# B&R Automation Studio project ACPtrak_Widget
Automation Studio 4.7.4.67 SP; technology packages: mappControl 5.11.0, mappMotion 5.11.2, mappView 5.11.2

## Configuration Simulation

CPU PC_any, AutomationRuntime A4.73, Build 4.1.2, Safety 0.0, Vc V4.62.0

### Task classes (Cpu.sw)
```
Cyclic#1 (cycle 400 us, tolerance 0 us):
  Main <- Main.prg
  WidgetData <- WidgetData.prg
Cyclic#2 (cycle 2000 us, tolerance 0 us):
  Vis <- Vis.prg
DataObjects: McAcpSys
Binaries: McAcpSim, FWRules, udbdef, McAcpDrv, arsvcreg, TCData, McProfGen, mvLoader, Config_1, Config_2, Config_4, ashwd, ashwac, asfw, iomap, sysconf, Config_3, Role, User, arconfig, Config_5, Config_6, Config_7, Config_8
Libraries: McBase, McAxis, McAcpTrak, McPureVAx, MpAxis, MpBase, TrakKit, standard, AsBrStr, McAcpAx, AsMath, FileIO, runtime, MTBasics, brsystem, MTTypes, sys_lib, powerlnk, astime, asieccon, arssl, asepl
```

### Hardware
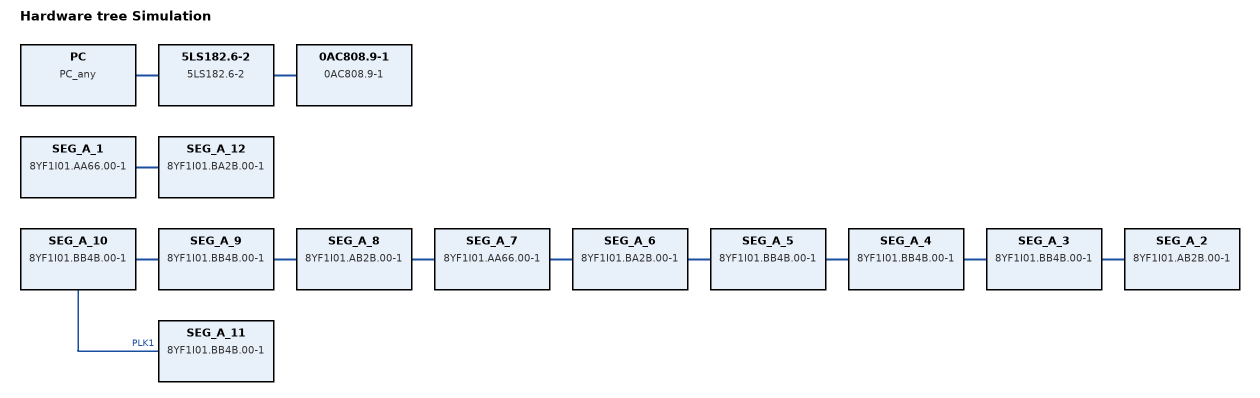
```
0AC808.9-1 : 0AC808.9-1 v1.0.0.0  [ETH1 -> 5LS182.6-2.IF1 [Cable Type=PowerlinkCable, Length=10, Version=1.0.0.2]; ETH2 -> SEG_A_1.PLK3 [Cable Type=PowerlinkCable, Length=10, Version=1.0.0.2]]
5LS182.6-2 : 5LS182.6-2 v1.4.0.0  [SL -> PC.SL2]
PC : PC_any v1.1.0.0 (OrderNumber=PC)
  ConfigurationID = StarwheelSim_Simulation
  VolatileGlobalPvSize = 132000
  SystemTick = 400
  Cyclic1Duration = 400
  Cyclic1Tolerance = 0
  Cyclic2Duration = 2000
  Cyclic2Tolerance = 0
  FileDevice1
  FileDeviceName1 = SvgData
  FileDevicePath1 = ../../../../Logical/Visuals
  FileDevice2
  FileDeviceName2 = User
  FileDevicePath2 = C:\ACPtrak\TeslaStarwheel\TrakPower
  ActivateOpcUa = 1
  OpcUaInformationModels_PV_Version = 1
SEG_A_1 : 8YF1I01.AA66.00-1 v0.0.0.3  [PLK1 -> SEG_A_2.PLK2 [Cable Type=PowerlinkCable, Length=10, Version=1.0.0.2]; PLK2 -> SEG_A_12.PLK1 [Cable Type=PowerlinkCable, Length=10, Version=1.0.0.2]; PLK3 -> 0AC808.9-1.ETH2 [Cable Type=PowerlinkCable, Length=10, Version=1.0.0.2]]
  DriveConfiguration:
    McTypeID = LLMConfig
  DriveConfiguration/Segment:
    Shape = STRAIGHT660
    SegmentReference = SEG_A_1
    StopReaction = UseAssemblySetting
    SpeedFilter = UseAssemblySetting
SEG_A_10 : 8YF1I01.BB4B.00-1 v0.0.0.3  [PLK1 -> SEG_A_11.PLK2 [Cable Type=PowerlinkCable, Length=10, Version=1.0.0.2]; PLK2 -> SEG_A_9.PLK1 [Cable Type=PowerlinkCable, Length=10, Version=1.0.0.2]]
  DriveConfiguration/Segment:
    SegmentReference = ::SEG_A_10
SEG_A_11 : 8YF1I01.BB4B.00-1 v0.0.0.3  [PLK2 -> SEG_A_10.PLK1 [Cable Type=PowerlinkCable, Length=10, Version=1.0.0.2]]
  DriveConfiguration/Segment:
    SegmentReference = ::SEG_A_11
SEG_A_12 : 8YF1I01.BA2B.00-1 v0.0.0.3  [PLK1 -> SEG_A_1.PLK2 [Cable Type=PowerlinkCable, Length=10, Version=1.0.0.2]]
  DriveConfiguration/Segment:
    SegmentReference = ::SEG_A_12
SEG_A_2 : 8YF1I01.AB2B.00-1 v0.0.0.3  [PLK1 -> SEG_A_3.PLK2 [Cable Type=PowerlinkCable, Length=10, Version=1.0.0.2]; PLK2 -> SEG_A_1.PLK1 [Cable Type=PowerlinkCable, Length=10, Version=1.0.0.2]]
  DriveConfiguration/Segment:
    SegmentReference = ::SEG_A_2
SEG_A_3 : 8YF1I01.BB4B.00-1 v0.0.0.3  [PLK1 -> SEG_A_4.PLK2 [Cable Type=PowerlinkCable, Length=10, Version=1.0.0.2]; PLK2 -> SEG_A_2.PLK1 [Cable Type=PowerlinkCable, Length=10, Version=1.0.0.2]]
  DriveConfiguration/Segment:
    SegmentReference = ::SEG_A_3
SEG_A_4 : 8YF1I01.BB4B.00-1 v0.0.0.3  [PLK1 -> SEG_A_5.PLK2 [Cable Type=PowerlinkCable, Length=10, Version=1.0.0.2]; PLK2 -> SEG_A_3.PLK1 [Cable Type=PowerlinkCable, Length=10, Version=1.0.0.2]]
  DriveConfiguration/Segment:
    SegmentReference = ::SEG_A_4
SEG_A_5 : 8YF1I01.BB4B.00-1 v0.0.0.3  [PLK1 -> SEG_A_6.PLK2 [Cable Type=PowerlinkCable, Length=10, Version=1.0.0.2]; PLK2 -> SEG_A_4.PLK1 [Cable Type=PowerlinkCable, Length=10, Version=1.0.0.2]]
  DriveConfiguration/Segment:
    SegmentReference = ::SEG_A_5
SEG_A_6 : 8YF1I01.BA2B.00-1 v0.0.0.3  [PLK1 -> SEG_A_7.PLK2 [Cable Type=PowerlinkCable, Length=10, Version=1.0.0.2]; PLK2 -> SEG_A_5.PLK1 [Cable Type=PowerlinkCable, Length=10, Version=1.0.0.2]]
  DriveConfiguration/Segment:
    SegmentReference = ::SEG_A_6
SEG_A_7 : 8YF1I01.AA66.00-1 v0.0.0.3  [PLK1 -> SEG_A_8.PLK2 [Cable Type=PowerlinkCable, Length=10, Version=1.0.0.2]; PLK2 -> SEG_A_6.PLK1 [Cable Type=PowerlinkCable, Length=10, Version=1.0.0.2]]
  DriveConfiguration/Segment:
    SegmentReference = ::SEG_A_7
SEG_A_8 : 8YF1I01.AB2B.00-1 v0.0.0.3  [PLK1 -> SEG_A_9.PLK2 [Cable Type=PowerlinkCable, Length=10, Version=1.0.0.2]; PLK2 -> SEG_A_7.PLK1 [Cable Type=PowerlinkCable, Length=10, Version=1.0.0.2]]
  DriveConfiguration/Segment:
    SegmentReference = ::SEG_A_8
SEG_A_9 : 8YF1I01.BB4B.00-1 v0.0.0.3  [PLK1 -> SEG_A_10.PLK2 [Cable Type=PowerlinkCable, Length=10, Version=1.0.0.2]; PLK2 -> SEG_A_8.PLK1 [Cable Type=PowerlinkCable, Length=10, Version=1.0.0.2]]
  DriveConfiguration/Segment:
    SegmentReference = ::SEG_A_9
```

### Config_1.assembly - PC/mappMotion/Config_1.assembly
```
Element gAssembly_1 (Type=assembly)
  Tracks:
    TrackSeparation = 0.030
    Track[1]:
      Segments:
        SegmentRef[1] = ::SEG_A_1
        SegmentRef[2] = ::SEG_A_2
        SegmentRef[3] = ::SEG_A_3
        SegmentRef[4] = ::SEG_A_4
        SegmentRef[5] = ::SEG_A_5
        SegmentRef[6] = ::SEG_A_6
        SegmentRef[7] = ::SEG_A_7
        SegmentRef[8] = ::SEG_A_8
        SegmentRef[9] = ::SEG_A_9
        SegmentRef[10] = ::SEG_A_10
        SegmentRef[11] = ::SEG_A_11
        SegmentRef[12] = ::SEG_A_12
      Position = Absolute
        SegmentCountDirection = RightToLeft
        Translation:
          X = 0.0
          Y = 0.0
          Z = 0.0
        Orientation:
          Angle1 = 0.0
          Angle2 = 0.0
          Angle3 = 180
  CommonSegmentSettings:
    SegmentSimulationOnPLC = Off
    StopReaction = InductionHalt
    SpeedFilter = NotUsed
    ControllerParameters:
      DefaultParameter:
        Controller:
          Position:
            ProportionalGain = 0.0
          Speed:
            ProportionalGain = 0.0
            IntegrationTime = 0.0
          FeedForward:
            TotalMass = 0.0
            ForcePositive = 0.0
            ForceNegative = 0.0
            SpeedForceFactor = 0.0
            ForceLoad = 0.0
        MovementErrorLimits:
          PositionError = 0.0
          VelocityError = 0.0
      AdditionalParameterSets = NotUsed
  Shuttles:
    MaxShuttleCount = 50
    ShuttleStereotypes:
      ShuttleStRef[1] = ShuttleStereotype_1
    MagnetPlateConfigurations:
      ShuttleType[1] = 8F1SA.102.xxxxxx-x
    CollisionAvoidance:
      Strategy = Constant
      MaximumModelDimensions:
        Length:
          ExtentToFront = 0.025
          ExtentToBack = 0.025
        Width:
          Width = 0.030
  Visualization:
    MonitoringPv = ::gShuttleMon
    ProcessingTaskClass = 2
```

### Config_2.shuttlestereotype - PC/mappMotion/Config_2.shuttlestereotype
```
Element ShuttleStereotype_1 (Type=shuttlestereotype)
  MeasurementUnit = 5067858
  MeasurementResolution = 0.00001
  MovementLimits = Internal
    VelocityIsReadOnly = 0
    Velocity:
      Velocity = 4.0
    AccelerationIsReadOnly = 0
    Acceleration:
      Acceleration = 50
    DecelerationIsReadOnly = 0
    Deceleration:
      Deceleration = 50
  JerkFilter = Used
    JerkTime = 0.02
  UserData:
    Size = 8
```

### Config_3.sector - PC/mappMotion/Config_3.sector
```
Element Sector_Spawn (Type=sector)
  Type = Composed
    StartSegment:
      SegmentRef = ::SEG_A_7
      Position = 0.33
      PositionRelativeTo = FromEnd
    EndSegment:
      SegmentRef = ::SEG_A_7
Element Sector_Infeed (Type=sector)
  Type = Composed
    StartSegment:
      SegmentRef = ::SEG_A_2
    IntermediateSegments:
      SegmentRef[1] = ::SEG_A_1
      SegmentRef[2] = ::SEG_A_12
      SegmentRef[3] = ::SEG_A_11
      SegmentRef[4] = ::SEG_A_10
      SegmentRef[5] = ::SEG_A_9
    EndSegment:
      SegmentRef = ::SEG_A_8
```

### Config_4.processpointlist - PC/mappMotion/Config_4.processpointlist
```
Element List_PP_Spawn (Type=processpointlist)
  ProcessPoint[0]:
    Name = PP_Spawn_In
    SectorRef = Sector_Spawn
    TriggerEventBufferSize = 10
    BarrierFunctionality = On
  ProcessPoint[1]:
    Name = PP_Spawn_Out
    SectorRef = Sector_Spawn
    PositionRelativeTo = FromEnd
    TriggerEventBufferSize = 10
    BarrierFunctionality = Off
Element List_PP_Outfeed (Type=processpointlist)
  ProcessPoint[0]:
    Name = PP_Outfeed_Sync
    SectorRef = Sector_Outfeed
    Position = 0.165
    TriggerEventBufferSize = 10
    BarrierFunctionality = Off
  ProcessPoint[1]:
    Name = PP_Outfeed_Release
    SectorRef = Sector_Outfeed
    Position = 0.57
    PositionRelativeTo = FromEnd
    TriggerEventBufferSize = 10
    BarrierFunctionality = Off
Element List_PP_Infeed (Type=processpointlist)
  ProcessPoint[0]:
    Name = PP_Infeed_Sync
    SectorRef = Sector_Infeed
    Position = 0.45
    TriggerEventBufferSize = 10
    BarrierFunctionality = On
  ProcessPoint[1]:
    Name = PP_Infeed_Release
    SectorRef = Sector_Infeed
    Position = 0.465
    PositionRelativeTo = FromEnd
    TriggerEventBufferSize = 10
    BarrierFunctionality = Off
```

### Config_5.axis - PC/mappMotion/InfeedAxis/Config_5.axis
```
Element gAxis_1 (Type=axis)
  BaseTypeIsReadOnly = 0
  BaseType = RotaryPeriodic
    MeasurementUnitIsReadOnly = 0
    MeasurementUnit = 17476
    MeasurementResolutionIsReadOnly = 0
    MeasurementResolution = 0.001
    CountDirectionIsReadOnly = 0
    CountDirection = Standard
    PeriodSettings:
      Period = 360.0
  MovementLimitsIsReadOnly = 0
  MovementLimits = Internal
    Position:
      LowerLimitMin = -1.79769313486231E308
      UpperLimitMax = 1.79769313486231E308
      LowerLimit = -1000.0
      UpperLimit = 1000.0
    VelocityIsReadOnly = 0
    Velocity:
      VelocityMax = 3.4E38
      Velocity = 720.0
    AccelerationIsReadOnly = 0
    Acceleration:
      AccelerationMax = 3.4E38
      Acceleration = 720.0
    DecelerationIsReadOnly = 0
    Deceleration:
      DecelerationMax = 3.4E38
      Deceleration = 720.0
  Alarms = None
```

### Config_6.purevaxcfg - PC/mappMotion/InfeedAxis/Config_6.purevaxcfg
```
Element PureVAxCfg_1 (Type=purevaxcfg)
  TypeID = PureVAxConfig
  PureVAxis:
    AxisReference = gAxis_1
```

## Logical view

Binary libraries used (declarations not repeated): operator, runtime, astime, AsIecCon, standard, AsBrStr, AsMath, FileIO, brsystem, MTTypes 1.03.4, sys_lib, McBase 5.11.2, McPureVAx 5.11.2, McAcpAx 5.11.2, McAcpTrak 5.11.2, McAxis 5.11.2, MpAxis 5.11.2, MpBase 5.11.0, MTBasics 5.11.0

### Global.typ - Global data types
```iecst
TYPE
	SyncObj_typ : 	STRUCT
		MoveCyclic : MC_BR_ElasticMoveCycPos_AcpTrak;
		InSync : BOOL;
		PocketSelect : USINT;
		ThisShuttle : McAxisType;
		PeriodSelect : USINT;
		LastCycleSetpoint : LREAL;
	END_STRUCT;
	UserData_typ : 	STRUCT
		SyncObjectID : UINT;
		Color : enumUserColor;
	END_STRUCT;
	TrakCmd_typ : 	STRUCT
		PowerOn : BOOL;
	END_STRUCT;
	TrakPar_typ : 	STRUCT
		Acceleration : REAL;
		Velocity : REAL;
		PPM : REAL;
	END_STRUCT;
	TrakStatus_typ : 	STRUCT
		State : USINT;
	END_STRUCT;
	Trak_typ : 	STRUCT
		Cmd : TrakCmd_typ;
		Par : TrakPar_typ;
		Status : TrakStatus_typ;
	END_STRUCT;
	Reference_typ : 	STRUCT
		PosRad : REAL;
		PosDeg : REAL;
	END_STRUCT;
	Period_typ : 	STRUCT
		Pocket : ARRAY[0..MAX_NUM_POCKETS]OF Pockets_typ;
		PocketLastCycle : ARRAY[0..MAX_NUM_POCKETS]OF Pockets_typ;
		TrakMax : REAL;
		TrakMin : REAL;
	END_STRUCT;
	Starwheel_typ : 	STRUCT
		Axis : MpAxisBasic;
		Period : ARRAY[0..MAX_NUM_PERIODS]OF Period_typ;
	END_STRUCT;
	Pockets_typ : 	STRUCT
		Offset : REAL;
		PosDeg : REAL;
		PosRad : REAL;
		TrakPos : LREAL;
	END_STRUCT;
	ProcessPoint_typ : 	STRUCT
		RoutedMoveVel : MC_BR_RoutedMoveVel_AcpTrak;
		TrgEnable : MC_BR_TrgPointEnable_AcpTrak;
		TrgInfo : MC_BR_TrgPointGetInfo_AcpTrak;
		ShUserData : MC_BR_ShCopyUserData_AcpTrak;
		UserDataBuffer : UserData_typ;
		Counter : UDINT;
		State : USINT;
		BarrierCmd : MC_BR_BarrierCommand_AcpTrak;
		BarrierReadInfo : MC_BR_BarrierReadInfo_AcpTrak;
		BarrierState : USINT;
		periodSelect : USINT;
		pocketSelect : USINT;
	END_STRUCT;
	StarSectorPar_typ : 	STRUCT
		R1 : REAL;
		R2 : REAL;
		deltaT : TIME;
		SectorTangentPos : REAL;
		PocketCount : USINT;
		Wm : REAL;
		ReleaseVelocity : REAL;
		PositionSyncPP : REAL;
		Rp : REAL;
		PeriodCount : USINT;
		PositionRelPP : REAL;
	END_STRUCT;
	StarwheelSectorLogic_typ : 	STRUCT
		Starwheel : Starwheel_typ;
		SyncPP : ProcessPoint_typ;
		ReleasePP : ProcessPoint_typ;
		SyncObj : ARRAY[0..NUM_SYNC_OBJS]OF SyncObj_typ;
		indexOpenSyncObj : USINT;
		Par : StarSectorPar_typ;
	END_STRUCT;
END_TYPE
```

### Segments.var - Global variables
```iecst
VAR
	SEG_A_1 : McSegmentType;
	SEG_A_2 : McSegmentType;
	SEG_A_3 : McSegmentType;
	SEG_A_4 : McSegmentType;
	SEG_A_5 : McSegmentType;
	SEG_A_6 : McSegmentType;
	SEG_A_7 : McSegmentType;
	SEG_A_8 : McSegmentType;
	SEG_A_9 : McSegmentType;
	SEG_A_10 : McSegmentType;
	SEG_A_11 : McSegmentType;
	SEG_A_12 : McSegmentType;
END_VAR
```

### Global.var - Global variables
```iecst
VAR
	gShuttleMon : McAcpTrakAssemblyMonData;
	gTrak : Trak_typ;
END_VAR
VAR CONSTANT
	NUM_SYNC_OBJS : USINT := 20;
	MAX_NUM_POCKETS : USINT := 16;
END_VAR
VAR
	Infeed : StarwheelSectorLogic_typ;
END_VAR
VAR CONSTANT
	MAX_NUM_PERIODS : USINT := 5;
END_VAR
```

### Package Logical/Libraries - Global libraries

### Library Logical/Libraries/TrakKit (IEC)

#### Types.typ - Exported data types
```iecst
TYPE
	enumUserColor :
		(
		GRAY,
		BLUE,
		RED,
		GREEN,
		YELLOW,
		ORANGE,
		WHITE,
		BLACK,
		PINK,
		PURPLE
		);
	typShuttleUserData : 	STRUCT
		Color : enumUserColor;
		SyncObjectID : UINT;
		InSync : BOOL;
	END_STRUCT;
	ClearBlockState :
		(
		CLEAR_BLOCK_STATE_IDLE,
		CLEAR_BLOCK_STATE_INIT,
		CLEAR_BLOCK_STATE_WAIT,
		CLEAR_BLOCK_STATE_RESET,
		CLEAR_BLOCK_STATE_OFF
		);
	ClearPPState :
		(
		CLEAR_PP_STATE_IDLE,
		CLEAR_PP_STATE_ENABLE,
		CLEAR_PP_STATE_WAIT,
		CLEAR_PP_STATE_GET_INFO,
		CLEAR_PP_STATE_OFF
		);
	SpawnState :
		(
		SPAWN_STATE_IDLE,
		SPAWN_STATE_BLOCK,
		SPAWN_STATE_CREATE,
		SPAWN_STATE_REPORT,
		SPAWN_STATE_CREATE_NEXT,
		SPAWN_STATE_GET,
		SPAWN_STATE_SET_USER_DATA,
		SPAWN_STATE_SEND,
		SPAWN_STATE_WAIT,
		SPAWN_STATE_TRIG,
		SPAWN_STATE_UNBLOCK,
		SPAWN_STATE_DONE
		);
	FeedState :
		(
		FEED_STATE_IDLE,
		FEED_STATE_ENABLE,
		FEED_STATE_WAIT,
		FEED_STATE_TRIG,
		FEED_STATE_CHECK_SHUTTLE,
		FEED_STATE_GET_SHUTTLE_DATA,
		FEED_STATE_MOVE_ABS,
		FEED_STATE_TIME,
		FEED_STATE_GET,
		FEED_STATE_COLOR,
		FEED_STATE_SEND,
		FEED_STATE_DISABLE
		);
	TwoUpState1 :
		(
		TWOUP_STATE1_IDLE,
		TWOUP_STATE1_ENABLE,
		TWOUP_STATE1_WAIT,
		TWOUP_STATE1_TRIG,
		TWOUP_STATE1_CHECK_SHUTTLE,
		TWOUP_STATE1_MOVE_ABS,
		TWOUP_STATE1_TIME,
		TWOUP_STATE1_DISABLE
		);
	TwoUpState2 :
		(
		TWOUP_STATE2_IDLE,
		TWOUP_STATE2_WAIT,
		TWOUP_STATE2_GET1,
		TWOUP_STATE2_MOVE_ABS,
		TWOUP_STATE2_TIME,
		TWOUP_STATE2_GET2,
		TWOUP_STATE2_COLOR,
		TWOUP_STATE2_SEND
		);
END_TYPE
```

#### TrakKit.fun - Exported functions and function blocks
```iecst
FUNCTION_BLOCK ShuttleSpawn
	VAR_INPUT
		Enable : BOOL;
		StartPP : UDINT; (*Process point at start to block any incoming shuttle*)
		EndPP : UDINT; (*Process point at end to check shuttles have left*)
		Sector : UDINT; (*Sector to create shuttles on*)
		SectorPositionStart : LREAL; (*Position to start creating shuttles*)
		SectorPositionIncrement : LREAL; (*Increment to create shuttles*)
		DstSector : DINT; (*Destination Sector*)
		DstSectorPosition : LREAL; (*Destination sector position*)
		Velocity : REAL; (*Velocity of move*)
		RouteVelocity : REAL;
		Acceleration : {REDUND_UNREPLICABLE} REAL; (*Acceleration of move*)
		NumShuttleBatch : USINT; (*Number of shuttles in a batch*)
		NumShuttleTotal : USINT; (*Total shuttles to spawn*)
		SetShuttleData : MC_BR_ShCopyUserData_AcpTrak;
		AcknSpawn : BOOL;
	END_VAR
	VAR_OUTPUT
		SpawnValid : BOOL;
		SpawnedAxis : McAxisType;
		Done : BOOL;
	END_VAR
	VAR
		InternalSectorPositionStart : LREAL;
		InternalSectorPositionIncrement : LREAL;
		InternalNumShuttleBatch : USINT;
		InternalNumShuttleTotal : USINT;
		ExitShuttleNum : USINT; (*Number of shuttles that have left*)
		BatchCreated : USINT; (*Number of shuttles created in the batch*)
		TotalCreated : USINT; (*Number of shuttles created total*)
		State : SpawnState;
		TrigEnable : MC_BR_TrgPointEnable_AcpTrak;
		TrigInfo : MC_BR_TrgPointGetInfo_AcpTrak;
		Barrier : MC_BR_BarrierCommand_AcpTrak;
		AddShuttle : MC_BR_SecAddShuttle_AcpTrak;
		GetShuttle : MC_BR_SecGetShuttle_AcpTrak;
		MoveVel : MC_BR_RoutedMoveVel_AcpTrak;
		InternalUserData : typShuttleUserData;
	END_VAR
END_FUNCTION_BLOCK

FUNCTION_BLOCK ShuttleDelete
END_FUNCTION_BLOCK

FUNCTION_BLOCK Redirect
END_FUNCTION_BLOCK

FUNCTION_BLOCK Feed
	VAR_INPUT
		Enable : BOOL;
		PP : UDINT;
		NumShuttles : USINT;
		Sector : UDINT;
		UseAbsMove : BOOL;
		UseVelMoveTrigger : BOOL;
		VelMovTrigger : BOOL;
		SectorPositionStart : LREAL;
		TrigDirection : McAcpTrakTrgPointEventEnum;
		MoveAbsVelocity : REAL;
		SectorPositionIncrement : LREAL;
		DstSector : UDINT;
		DstSectorPosition : LREAL;
		DstStartDirection : McDirectionEnum;
		Color : enumUserColor;
		Velocity : REAL;
		RouteVelocity : REAL;
		Acceleration : REAL;
		FeedTime : TIME;
	END_VAR
	VAR_OUTPUT
		Done : BOOL;
		ReadyForProduct : BOOL;
	END_VAR
	VAR
		InternalNumShuttles : USINT;
		InternalSectorPositionStart : LREAL;
		InternalSectorPositionIncrement : LREAL;
		InternalUserData : typShuttleUserData;
		LastSeqNumber : UDINT;
		LastShuttleNumber : USINT;
		ShuttleCount : USINT;
		State : FeedState;
		TrigEnable : MC_BR_TrgPointEnable_AcpTrak;
		TrigInfo : MC_BR_TrgPointGetInfo_AcpTrak;
		CheckShuttle : MC_BR_ShReadInfo_AcpTrak;
		MoveAbs : MC_BR_RoutedMoveAbs_AcpTrak;
		GetShuttle : MC_BR_SecGetShuttle_AcpTrak;
		ColorShuttle : MC_BR_ShCopyUserData_AcpTrak;
		MoveVel : MC_BR_RoutedMoveVel_AcpTrak;
		FeedTON : TON;
		ReadShuttleData : MC_BR_ShCopyUserData_AcpTrak;
	END_VAR
END_FUNCTION_BLOCK

FUNCTION_BLOCK ClearArea
	VAR_INPUT
		Enable : BOOL;
		StartPP : UDINT;
		EndPP : UDINT;
		NumShuttles : USINT; (*Number of shuttles to allow*)
		newParam : BOOL;
	END_VAR
	VAR
		ExitShuttleNum : USINT; (*Number of shuttles that have left*)
		BlockState : ClearBlockState;
		PPState : ClearPPState;
		TrigEnable : MC_BR_TrgPointEnable_AcpTrak;
		TrigInfo : MC_BR_TrgPointGetInfo_AcpTrak;
		Barrier : MC_BR_BarrierCommand_AcpTrak;
	END_VAR
END_FUNCTION_BLOCK

FUNCTION_BLOCK CalculatePPM
	VAR_INPUT
		Enable : BOOL;
		PP : UDINT;
		NumberOfShuttlesToAvg : LREAL; (*Max 10000*)
		TrigDirection : McAcpTrakTrgPointEventEnum;
	END_VAR
	VAR_OUTPUT
		PPM : LREAL;
	END_VAR
	VAR
		FinishedLoadout : BOOL;
		LastSeqNumber : UDINT;
		ShuttlesPassed : INT;
		TotalShuttlesPassed : UDINT;
		TimeTotal : UDINT;
		TimeStart : ARRAY[0..10000] OF DATE_AND_TIME;
		TimeDelta : UDINT;
		State : UINT;
		TrigEnable : MC_BR_TrgPointEnable_AcpTrak;
		TrigInfo : MC_BR_TrgPointGetInfo_AcpTrak;
		CheckShuttle : MC_BR_ShReadInfo_AcpTrak;
		DTGetTime_0 : DTGetTime;
		LastTimeDeltaIndex : UINT;
	END_VAR
END_FUNCTION_BLOCK

FUNCTION_BLOCK TwoUp
	VAR_INPUT
		Enable : BOOL;
		PP : UDINT;
		NumShuttles : USINT;
		Sector : ARRAY[0..1] OF UDINT;
		SectorPositionStart : ARRAY[0..1] OF LREAL;
		SectorPositionIncrement : ARRAY[0..1] OF LREAL;
		DstSector : UDINT;
		DstSectorPosition : LREAL;
		Color : enumUserColor;
		Velocity : REAL;
		Acceleration : REAL;
		FeedTime : ARRAY[0..1] OF TIME;
	END_VAR
	VAR
		InternalNumShuttles : USINT;
		InternalPosArray : ARRAY[0..8] OF LREAL;
		InternalSectorPositionStart : ARRAY[0..1] OF LREAL;
		InternalSectorPositionIncrement : ARRAY[0..1] OF LREAL;
		InternalUserData : typShuttleUserData;
		ShuttleCount : USINT;
		State1 : TwoUpState1;
		State2 : TwoUpState2;
		TrigEnable : MC_BR_TrgPointEnable_AcpTrak;
		TrigInfo : MC_BR_TrgPointGetInfo_AcpTrak;
		CheckShuttle : MC_BR_ShReadInfo_AcpTrak;
		MoveAbs : ARRAY[0..1] OF MC_BR_RoutedMoveAbs_AcpTrak;
		GetShuttle : ARRAY[0..1] OF MC_BR_SecGetShuttle_AcpTrak;
		MoveVel : MC_BR_RoutedMoveVel_AcpTrak;
		ColorShuttle : MC_BR_ShCopyUserData_AcpTrak;
		FeedTON : ARRAY[0..1] OF TON;
		Increment : BOOL; (*Increment from first to second segment*)
	END_VAR
END_FUNCTION_BLOCK
```

#### ShuttleSpawn.st
```iecst
FUNCTION_BLOCK ShuttleSpawn

	CASE State OF

		SPAWN_STATE_IDLE:

			IF Enable THEN
				InternalSectorPositionStart := SectorPositionStart;
				InternalSectorPositionIncrement := SectorPositionIncrement;
				InternalNumShuttleTotal := NumShuttleTotal;
				InternalNumShuttleBatch := NumShuttleBatch;
				//				InternalUserData.ShuttleNumber := 0;
				//				InternalUserData.Color := BLUE;
			//	InternalUserData.FirstShuttle := 1;
				TrigEnable.ProcessPoint := EndPP;
				TrigEnable.Enable := 1;
				TrigInfo.ProcessPoint := EndPP;
				Barrier.ProcessPoint := StartPP;
				Barrier.Command := mcACPTRAK_BARRIER_CLOSE;
				Barrier.Execute := 1;
				AddShuttle.Sector := Sector;
				AddShuttle.AdvancedParameters.Velocity := Velocity;
				AddShuttle.Position := InternalSectorPositionStart;
				GetShuttle.Sector := Sector;
				GetShuttle.Mode := mcACPTRAK_SEARCH_FORWARD;
//  added F.Forthuber
				SpawnValid := FALSE;
//  end
				SetShuttleData.Axis  := ADR(GetShuttle.Axis);
				SetShuttleData.DataAddress := ADR(InternalUserData);
				SetShuttleData.DataSize := SIZEOF(InternalUserData);
				SetShuttleData.Mode := mcACPTRAK_USERDATA_SET;
				MoveVel.Axis := ADR(GetShuttle.Axis);
				MoveVel.Sector := DstSector;
				MoveVel.Position := DstSectorPosition;
				MoveVel.Velocity := Velocity;
				MoveVel.RouteVelocity := RouteVelocity;
				MoveVel.Acceleration := Acceleration;
				MoveVel.Deceleration := Acceleration;
				MoveVel.AdvancedParameters.StartDirection := mcDIR_POSITIVE;
				MoveVel.AdvancedParameters.EndDirection := mcDIR_POSITIVE;
				MoveVel.AdvancedParameters.ShuttleOrientation := mcDIR_UNDEFINED;
				State := SPAWN_STATE_BLOCK;
			END_IF

		SPAWN_STATE_BLOCK:

			IF TrigEnable.Valid AND Barrier.Done THEN
				Barrier.Execute := 0;
				AddShuttle.Execute := 1;
				Done:=FALSE;
				State := SPAWN_STATE_CREATE;
			END_IF

		SPAWN_STATE_CREATE:

			IF AddShuttle.Done THEN
//  added F.Forthuber
				SpawnedAxis := AddShuttle.Axis;
				SpawnValid:=TRUE;
				State := SPAWN_STATE_REPORT;
			END_IF

		SPAWN_STATE_REPORT:

			IF AcknSpawn THEN
				SpawnValid:=FALSE;
//  end
				BatchCreated := BatchCreated + 1;
				TotalCreated := TotalCreated + 1;
				AddShuttle.Execute := 0;
				IF (BatchCreated >= InternalNumShuttleBatch) OR (TotalCreated >= InternalNumShuttleTotal) THEN
					BatchCreated := 0;
					GetShuttle.Enable := 1;
					State := SPAWN_STATE_GET;
				ELSE
					State := SPAWN_STATE_CREATE_NEXT;
				END_IF
			END_IF

		SPAWN_STATE_CREATE_NEXT:

			AddShuttle.Position := AddShuttle.Position + InternalSectorPositionIncrement;
			AddShuttle.Execute := 1;
			State := SPAWN_STATE_CREATE;

		SPAWN_STATE_GET:

			IF GetShuttle.Valid THEN
				GetShuttle.Next := 0;
				//InternalUserData.ShuttleNumber := InternalUserData.ShuttleNumber + 1;
				SetShuttleData.Execute := 1;
				State := SPAWN_STATE_SET_USER_DATA;
			END_IF

		SPAWN_STATE_SET_USER_DATA:
			IF SetShuttleData.Done THEN
				SetShuttleData.Execute := 0;
				MoveVel.Execute := 1;
				State := SPAWN_STATE_SEND;
			END_IF;

		SPAWN_STATE_SEND:

			IF MoveVel.Active THEN
	//			InternalUserData.FirstShuttle := 0;
				MoveVel.Execute := 0;
				IF GetShuttle.RemainingCount = 0 THEN
					GetShuttle.Enable := 0;
					State := SPAWN_STATE_WAIT;
				ELSE
					GetShuttle.Next := 1;
					State := SPAWN_STATE_GET;
				END_IF
			END_IF

		SPAWN_STATE_WAIT:

			IF NOT Enable  THEN
				TotalCreated := 0;
				ExitShuttleNum := 0;
				TrigEnable.Enable := 0;
				Barrier.Command := mcACPTRAK_BARRIER_OPEN;
				Barrier.Execute := 1;
				State := SPAWN_STATE_UNBLOCK;
			ELSIF TotalCreated >= InternalNumShuttleTotal THEN
				TotalCreated := 0;
				TrigEnable.Enable := 0;
				Barrier.Command := mcACPTRAK_BARRIER_OPEN;
				Barrier.Execute := 1;
				State := SPAWN_STATE_UNBLOCK;
			ELSIF ExitShuttleNum >= InternalNumShuttleBatch THEN
				ExitShuttleNum := 0;
				AddShuttle.Position := InternalSectorPositionStart;
				AddShuttle.Execute := 1;
				State := SPAWN_STATE_CREATE;
			ELSIF TrigEnable.EventCount > 0 THEN
				TrigInfo.Execute := 1;
				State := SPAWN_STATE_TRIG;
			END_IF

		SPAWN_STATE_TRIG:

			IF TrigInfo.Done THEN
				TrigInfo.Execute := 0;
				ExitShuttleNum := ExitShuttleNum + 1;
				State := SPAWN_STATE_WAIT;
			END_IF

		SPAWN_STATE_UNBLOCK:

			IF Barrier.Done AND NOT TrigEnable.Valid THEN
				Barrier.Execute := 0;
				State := SPAWN_STATE_DONE;
			END_IF

		SPAWN_STATE_DONE:

			Done := TRUE;

			IF NOT Enable THEN
				Done := FALSE;
				State := SPAWN_STATE_IDLE;
			END_IF

	END_CASE

	TrigEnable();
	TrigInfo();
	Barrier();
	AddShuttle();
	GetShuttle();
	SetShuttleData();
	MoveVel();

END_FUNCTION_BLOCK
```

#### ShuttleDelete.st
```iecst
FUNCTION_BLOCK ShuttleDelete

END_FUNCTION_BLOCK
```

#### Redirect.st
```iecst
FUNCTION_BLOCK Redirect

(*)
Redirect.st

IF Redirect.ShuttlePassed AND Redirect.ShuttleInfoValid THEN

	CASE Redirect.ShuttleInfo OF

	Redirect.DestinationSector		:= SECTOR_A;
	Redirect.DestinationPosition	:= 3.0;
	Redirect.Velocity				:= whatver;
	Redirect.Accel					:= whatever

	Redirect.Execute				:= TRUE;
ELSE
	Redirect.Execute				:= FALSE;
END_IF;
*)

END_FUNCTION_BLOCK
```

#### Feed.st
```iecst
FUNCTION_BLOCK Feed

	CASE State OF

		FEED_STATE_IDLE:

			IF Enable THEN
				InternalNumShuttles := NumShuttles;
				InternalSectorPositionStart := SectorPositionStart;
				InternalSectorPositionIncrement := SectorPositionIncrement;
				TrigEnable.ProcessPoint := PP;
				TrigEnable.Enable := 1;
				TrigInfo.ProcessPoint := PP;
				CheckShuttle.Axis := ADR(TrigInfo.TrgPointInfo.Axis);
				MoveAbs.Axis := ADR(TrigInfo.TrgPointInfo.Axis);
				MoveAbs.Sector := Sector;
				MoveAbs.Position := InternalSectorPositionStart;
				MoveAbs.Velocity := MoveAbsVelocity;
				MoveAbs.Acceleration := Acceleration;
				MoveAbs.Deceleration := Acceleration;
				MoveAbs.AdvancedParameters.StartDirection := mcDIR_POSITIVE;
				MoveAbs.AdvancedParameters.EndDirection := mcDIR_UNDEFINED;
				MoveAbs.AdvancedParameters.ShuttleOrientation := mcDIR_UNDEFINED;
				FeedTON.PT := FeedTime;
				GetShuttle.Sector := Sector;
				GetShuttle.Mode :=  mcACPTRAK_SEARCH_BACKWARD;
				ColorShuttle.Axis  := ADR(GetShuttle.Axis);
				ColorShuttle.DataAddress := ADR(InternalUserData);
				ColorShuttle.DataSize := SIZEOF(InternalUserData);
				ColorShuttle.Mode := mcACPTRAK_USERDATA_SET;
				ReadShuttleData.Axis  := ADR(TrigInfo.TrgPointInfo.Axis);
				ReadShuttleData.DataAddress := ADR(InternalUserData);
				ReadShuttleData.DataSize := SIZEOF(InternalUserData);
				ReadShuttleData.Mode := mcACPTRAK_USERDATA_GET;
				MoveVel.Axis := ADR(GetShuttle.Axis);
				MoveVel.Sector := DstSector;
				MoveVel.Position := DstSectorPosition;
				MoveVel.Velocity := Velocity;
				MoveVel.RouteVelocity := RouteVelocity;
				MoveVel.Acceleration := Acceleration;
				MoveVel.Deceleration := Acceleration;
				MoveVel.AdvancedParameters.StartDirection := DstStartDirection;// mcDIR_NEGATIVE;
				MoveVel.AdvancedParameters.EndDirection := mcDIR_UNDEFINED;
				MoveVel.AdvancedParameters.ShuttleOrientation := mcDIR_UNDEFINED;
				State := FEED_STATE_ENABLE;
			END_IF

		FEED_STATE_ENABLE:

			IF TrigEnable.Valid THEN
				State := FEED_STATE_WAIT;
			END_IF

		FEED_STATE_WAIT:

			IF ShuttleCount = 0 AND NOT Enable THEN
				TrigEnable.Enable := 0;
				State := FEED_STATE_DISABLE;
			ELSIF TrigEnable.EventCount > 0 THEN
				TrigInfo.Execute := 1;
				State := FEED_STATE_TRIG;
			END_IF

		FEED_STATE_TRIG:

			IF TrigInfo.Done THEN
				IF TrigInfo.TrgPointInfo.Event = TrigDirection THEN  // mcACPTRAK_TP_PASSED_POSITIVE THEN
					MoveVel.Velocity := Velocity;
					MoveVel.RouteVelocity := RouteVelocity;
					MoveAbs.Velocity := MoveAbsVelocity;

					CheckShuttle.Enable := 1;
					State := FEED_STATE_CHECK_SHUTTLE;
				ELSE
					TrigInfo.Execute := 0;
					State := FEED_STATE_WAIT;
				END_IF
			END_IF

		FEED_STATE_CHECK_SHUTTLE:

			IF CheckShuttle.Valid AND TrigInfo.TrgPointInfo.Axis.seqNo <> LastSeqNumber THEN // (CheckShuttle.ShuttleInfo.CurrentValues.SectorType <> mcACPTRAK_SEC_INTERNAL) THEN //
				LastSeqNumber := TrigInfo.TrgPointInfo.Axis.seqNo;
				Done:=FALSE;
				ShuttleCount := ShuttleCount + 1;
				ReadShuttleData.Execute := 1;
				IF UseAbsMove THEN
					//MoveAbs.Position := InternalSectorPositionStart;
					MoveAbs.Execute := 1;
					State := FEED_STATE_MOVE_ABS;
				ELSE
					GetShuttle.Enable := 1;
					State := FEED_STATE_GET;
				END_IF
			ELSE
				CheckShuttle.Enable := 0;
				TrigInfo.Execute := 0;
				State := FEED_STATE_WAIT;
			END_IF

		FEED_STATE_GET_SHUTTLE_DATA:
			IF ReadShuttleData.Done THEN
		//		LastShuttleNumber := InternalUserData.ShuttleNumber;
				IF UseAbsMove THEN
					MoveAbs.Execute := 1;
					State := FEED_STATE_MOVE_ABS;
				ELSE
					GetShuttle.Enable := 1;
					State := FEED_STATE_GET;
				END_IF

			ELSE
				State := FEED_STATE_WAIT;
			END_IF

		FEED_STATE_MOVE_ABS:
			ReadShuttleData.Execute := FALSE;
			IF MoveAbs.Active THEN
				IF ShuttleCount < InternalNumShuttles THEN
					MoveAbs.Execute := 0;
					CheckShuttle.Enable := 0;
					TrigInfo.Execute := 0;
					MoveAbs.Position := MoveAbs.Position - InternalSectorPositionIncrement;
					State := FEED_STATE_WAIT;
				END_IF
			ELSIF MoveAbs.Done THEN  // OR CheckShuttle.ShuttleInfo.CurrentValues.Velocity < 0.01 THEN
				MoveAbs.Execute := 0;
				CheckShuttle.Enable := 0;
				TrigInfo.Execute := 0;
				IF ShuttleCount >= InternalNumShuttles THEN
					ShuttleCount := 0;
					MoveAbs.Position := InternalSectorPositionStart;
					FeedTON.IN := 1;
					State := FEED_STATE_TIME;
				ELSE
					MoveAbs.Position := MoveAbs.Position - InternalSectorPositionIncrement;
					State := FEED_STATE_WAIT;
				END_IF
			END_IF

		FEED_STATE_TIME:
			ReadyForProduct := TRUE;
			IF FeedTON.Q THEN
				FeedTON.IN := 0;
				GetShuttle.Enable := 1;
				State := FEED_STATE_GET;
			END_IF

		FEED_STATE_GET:

			IF GetShuttle.Valid THEN
				GetShuttle.Next := 0;
				InternalUserData.Color := Color;
	//			InternalUserData.ShuttleNumber := LastShuttleNumber;
				ColorShuttle.Execute := 1;
				State := FEED_STATE_COLOR;
			END_IF

		FEED_STATE_COLOR:
			IF ColorShuttle.Done THEN
				ColorShuttle.Execute := 0;
				MoveVel.Execute := 1;
				State := FEED_STATE_SEND;
				ReadyForProduct:=FALSE;
			END_IF;
		FEED_STATE_SEND:

			IF MoveVel.Active THEN
				MoveVel.Execute := 0;
				Done:=TRUE;
				IF GetShuttle.RemainingCount = 0 THEN
					GetShuttle.Enable := 0;
					State := FEED_STATE_WAIT;
				ELSE
					GetShuttle.Next := 1;
					State := FEED_STATE_GET;
				END_IF
			END_IF

		FEED_STATE_DISABLE:

			IF NOT TrigEnable.Valid THEN
				State := FEED_STATE_IDLE;
			END_IF

	END_CASE

	TrigEnable();
	TrigInfo();
	CheckShuttle();
	MoveAbs();
	GetShuttle();
	ColorShuttle();
	MoveVel();
	FeedTON();
	ReadShuttleData();

END_FUNCTION_BLOCK
```

#### ClearArea.st
```iecst
FUNCTION_BLOCK ClearArea

	CASE BlockState OF

		CLEAR_BLOCK_STATE_IDLE:

			IF Enable THEN
				Barrier.ProcessPoint := StartPP;
				Barrier.AdvancedParameters.TicketCount := NumShuttles;
				Barrier.Command := mcACPTRAK_BARRIER_ADD_TICKETS;
				Barrier.Execute := 1;
				BlockState := CLEAR_BLOCK_STATE_INIT;
			END_IF

		CLEAR_BLOCK_STATE_INIT:

			IF Barrier.Done THEN
				Barrier.Execute := 0;
				BlockState := CLEAR_BLOCK_STATE_WAIT;
			END_IF

		CLEAR_BLOCK_STATE_WAIT:

			IF NOT Enable THEN
				Barrier.AdvancedParameters.TicketCount := 0;
				Barrier.Command := mcACPTRAK_BARRIER_OPEN;
				Barrier.Execute := 1;
				BlockState := CLEAR_BLOCK_STATE_OFF;
			ELSIF USINT_TO_DINT(ExitShuttleNum) >= Barrier.AdvancedParameters.TicketCount THEN
				ExitShuttleNum := 0;
				Barrier.Execute := 1;
				BlockState := CLEAR_BLOCK_STATE_RESET;
			END_IF

		CLEAR_BLOCK_STATE_RESET:

			IF Barrier.Done THEN
				Barrier.Execute := 0;
				BlockState := CLEAR_BLOCK_STATE_WAIT;
			END_IF

		CLEAR_BLOCK_STATE_OFF:

			IF Barrier.Done THEN
				ExitShuttleNum := 0;
				Barrier.Execute := 0;
				BlockState := CLEAR_BLOCK_STATE_IDLE;
			END_IF

	END_CASE

	CASE PPState OF

		CLEAR_PP_STATE_IDLE:

			IF Enable THEN
				TrigEnable.ProcessPoint := EndPP;
				TrigEnable.Enable := 1;
				TrigInfo.ProcessPoint := EndPP;
				PPState := CLEAR_PP_STATE_ENABLE;
			END_IF

		CLEAR_PP_STATE_ENABLE:

			IF TrigEnable.Valid THEN
				PPState := CLEAR_PP_STATE_WAIT;
			END_IF

		CLEAR_PP_STATE_WAIT:

			IF NOT Enable THEN
				TrigEnable.Enable := 0;
				PPState := CLEAR_PP_STATE_OFF;
			ELSIF TrigEnable.EventCount > 0  THEN
				TrigInfo.Execute := 1;
				PPState := CLEAR_PP_STATE_GET_INFO;
			END_IF

		CLEAR_PP_STATE_GET_INFO:

			IF TrigInfo.Done THEN
				ExitShuttleNum := ExitShuttleNum + 1;
				TrigInfo.Execute := 0;
				PPState := CLEAR_PP_STATE_WAIT;
			END_IF

		CLEAR_PP_STATE_OFF:

			IF NOT TrigEnable.Valid THEN
				ExitShuttleNum := 0;
				PPState := CLEAR_PP_STATE_IDLE;
			END_IF

	END_CASE

	TrigEnable();
	TrigInfo();
	Barrier();
END_FUNCTION_BLOCK
```

#### CalcPPM.st
```iecst
FUNCTION_BLOCK CalculatePPM

	CASE State OF

		0:

			IF Enable THEN
				TrigEnable.ProcessPoint := PP;
				TrigEnable.Enable := TRUE;
				TrigInfo.ProcessPoint := PP;
				CheckShuttle.Axis := ADR(TrigInfo.TrgPointInfo.Axis);
				DTGetTime_0.enable := TRUE;
				State := 1;
				//ShuttlesPassed:=1;
			END_IF

		1:
			//TotalShuttlesPassed := 0;
			IF TrigEnable.Valid THEN
				State := 2;
			END_IF

		2:

			IF NOT Enable THEN
				TrigEnable.Enable := FALSE;
			ELSIF TrigEnable.EventCount > 0 THEN
				IF NumberOfShuttlesToAvg > 10000 THEN
					NumberOfShuttlesToAvg:=10000;
				END_IF
				TrigInfo.Execute := TRUE;
				State := 3;
			END_IF

		3:

			IF TrigInfo.Done THEN
				IF TrigInfo.TrgPointInfo.Event = TrigDirection THEN
					CheckShuttle.Enable := TRUE;
					State := 4;
				ELSE
					TrigInfo.Execute := 0;
					State := 2;
				END_IF
			END_IF

		4:

			IF CheckShuttle.Valid AND TrigInfo.TrgPointInfo.Axis.seqNo <> LastSeqNumber THEN
				LastSeqNumber := TrigInfo.TrgPointInfo.Axis.seqNo;

				IF TotalShuttlesPassed = 0 THEN
					TimeStart[0] := DTGetTime_0.DT1;
				ELSE
					ShuttlesPassed := ShuttlesPassed + 1;
					IF ShuttlesPassed > NumberOfShuttlesToAvg THEN
						ShuttlesPassed := 1;
					END_IF;
					IF TotalShuttlesPassed <= NumberOfShuttlesToAvg THEN
						TimeStart[ShuttlesPassed]:=DTGetTime_0.DT1;
						TimeDelta := DiffDT(DTGetTime_0.DT1, TimeStart[0]);
						PPM := 60.0 * INT_TO_LREAL(ShuttlesPassed) / UDINT_TO_LREAL(TimeDelta);
						//LastTimeDeltaIndex:=1;
					ELSE
						//						LastTimeDeltaIndex:=LastTimeDeltaIndex+1;
						//						IF LastTimeDeltaIndex > NumberOfShuttlesToAvg THEN
						//							LastTimeDeltaIndex:=1;
						//						END_IF;
						TimeDelta := DiffDT(DTGetTime_0.DT1, TimeStart[ShuttlesPassed]);
						TimeStart[ShuttlesPassed]:=DTGetTime_0.DT1;
						PPM := 60.0 * NumberOfShuttlesToAvg / UDINT_TO_LREAL(TimeDelta);
					END_IF
				END_IF
				TotalShuttlesPassed := TotalShuttlesPassed +1;

			END_IF
			CheckShuttle.Enable := 0;
			TrigInfo.Execute := 0;
			State := 2;

	END_CASE

	TrigEnable();
	TrigInfo();
	CheckShuttle();
	DTGetTime_0();

END_FUNCTION_BLOCK
```

#### TwoUp.st
```iecst
FUNCTION_BLOCK TwoUp

	CASE State1 OF

		TWOUP_STATE1_IDLE:

			IF Enable THEN
				InternalNumShuttles := NumShuttles;

				InternalPosArray[0] := 0.80;
				InternalPosArray[1] := 0.72;
				InternalPosArray[2] := 0.64;
				InternalPosArray[3] := 0.56;
				InternalPosArray[4] := 0.32;
				InternalPosArray[5] := 0.24;
				InternalPosArray[6] := 0.16;
				InternalPosArray[7] := 0.08;

				InternalSectorPositionStart[0] := SectorPositionStart[0];
				InternalSectorPositionIncrement[0] := SectorPositionIncrement[0];
				TrigEnable.ProcessPoint := PP;
				TrigEnable.Enable := 1;
				TrigInfo.ProcessPoint := PP;
				CheckShuttle.Axis := ADR(TrigInfo.TrgPointInfo.Axis);
				MoveAbs[0].Axis := ADR(TrigInfo.TrgPointInfo.Axis);
				MoveAbs[0].Sector := Sector[0];

				MoveAbs[0].Position := (*InternalPosArray[1];//*)InternalSectorPositionStart[0];

				MoveAbs[0].Velocity := Velocity;
				MoveAbs[0].Acceleration := Acceleration;
				MoveAbs[0].Deceleration := Acceleration;
				MoveAbs[0].AdvancedParameters.StartDirection := mcDIR_POSITIVE;
				MoveAbs[0].AdvancedParameters.EndDirection := mcDIR_UNDEFINED;
				MoveAbs[0].AdvancedParameters.ShuttleOrientation := mcDIR_UNDEFINED;
				FeedTON[0].PT := FeedTime[0];
				State1 := TWOUP_STATE1_ENABLE;
			END_IF

		TWOUP_STATE1_ENABLE:

			IF TrigEnable.Valid THEN
				State1 := TWOUP_STATE1_WAIT;
			END_IF

		TWOUP_STATE1_WAIT:

			IF ShuttleCount = 0 AND NOT Enable THEN
				TrigEnable.Enable := 0;
				State1 := TWOUP_STATE1_DISABLE;
			ELSIF TrigEnable.EventCount > 0 THEN
				TrigInfo.Execute := 1;
				State1 := TWOUP_STATE1_TRIG;
			END_IF

		TWOUP_STATE1_TRIG:

			IF TrigInfo.Done THEN
				CheckShuttle.Enable := 1;
				State1 := TWOUP_STATE1_CHECK_SHUTTLE;
			END_IF

		TWOUP_STATE1_CHECK_SHUTTLE:

			IF CheckShuttle.Valid AND (CheckShuttle.ShuttleInfo.CurrentValues.SectorType <> mcACPTRAK_SEC_INTERNAL) THEN
				ShuttleCount := ShuttleCount + 1;
				MoveAbs[0].Execute := 1;
				State1 := TWOUP_STATE1_MOVE_ABS;
			ELSE
				CheckShuttle.Enable := 0;
				TrigInfo.Execute := 0;
				State1 := TWOUP_STATE1_WAIT;
			END_IF

		TWOUP_STATE1_MOVE_ABS:

			IF MoveAbs[0].Active THEN
				IF ShuttleCount < InternalNumShuttles THEN
					MoveAbs[0].Execute := 0;
					CheckShuttle.Enable := 0;
					TrigInfo.Execute := 0;
					MoveAbs[0].Position := (*InternalPosArray[ShuttleCount];//*)MoveAbs[0].Position - InternalSectorPositionIncrement[0];
					State1 := TWOUP_STATE1_WAIT;
				END_IF
			ELSIF MoveAbs[0].Done THEN
				MoveAbs[0].Execute := 0;
				CheckShuttle.Enable := 0;
				TrigInfo.Execute := 0;
				IF ShuttleCount >= InternalNumShuttles THEN
					ShuttleCount := 0;
					MoveAbs[0].Position := (*InternalPosArray[1];//*)InternalSectorPositionStart[0];
					FeedTON[0].IN := 1;
					State1 := TWOUP_STATE1_TIME;
				ELSE
					MoveAbs[0].Position := (*InternalPosArray[ShuttleCount];//*)MoveAbs[0].Position - InternalSectorPositionIncrement[0];
					State1 := TWOUP_STATE1_WAIT;
				END_IF
			END_IF

		TWOUP_STATE1_TIME:

			IF FeedTON[0].Q THEN
				FeedTON[0].IN := 0;
				Increment := 1;
				State1 := TWOUP_STATE1_WAIT;
			END_IF

		TWOUP_STATE1_DISABLE:

			IF NOT TrigEnable.Valid THEN
				State1 := TWOUP_STATE1_IDLE;
			END_IF

	END_CASE

	CASE State2 OF

		TWOUP_STATE2_IDLE:

			IF Enable THEN
				Increment := 0;
				InternalSectorPositionStart[1] := SectorPositionStart[1];
				InternalSectorPositionIncrement[1] := SectorPositionIncrement[1];
				InternalUserData.Color := Color;
				GetShuttle[0].Sector := Sector[0];
				GetShuttle[0].Mode :=  mcACPTRAK_SEARCH_BACKWARD;
				MoveAbs[1].Axis := ADR(GetShuttle[0].Axis);
				MoveAbs[1].Sector := Sector[1];
				MoveAbs[1].Position := InternalSectorPositionStart[1];
				MoveAbs[1].Velocity := Velocity;
				MoveAbs[1].Acceleration := Acceleration;
				MoveAbs[1].Deceleration := Acceleration;
				MoveAbs[1].AdvancedParameters.StartDirection := mcDIR_POSITIVE;
				MoveAbs[1].AdvancedParameters.EndDirection := mcDIR_UNDEFINED;
				MoveAbs[1].AdvancedParameters.ShuttleOrientation := mcDIR_UNDEFINED;
				FeedTON[1].PT := FeedTime[1];
				GetShuttle[1].Sector := Sector[1];
				GetShuttle[1].Mode :=  mcACPTRAK_SEARCH_FORWARD;
				ColorShuttle.Axis  := ADR(GetShuttle[1].Axis);
				ColorShuttle.DataAddress := ADR(InternalUserData);
				ColorShuttle.DataSize := SIZEOF(InternalUserData);
				ColorShuttle.Mode := mcACPTRAK_USERDATA_SET;
				MoveVel.Axis := ADR(GetShuttle[1].Axis);
				MoveVel.Sector := DstSector;
				MoveVel.Position := DstSectorPosition;
				MoveVel.Velocity := Velocity;
				MoveVel.RouteVelocity := Velocity;
				MoveVel.Acceleration := Acceleration;
				MoveVel.Deceleration := Acceleration;
				MoveVel.AdvancedParameters.StartDirection := mcDIR_POSITIVE;
				MoveVel.AdvancedParameters.EndDirection := mcDIR_UNDEFINED;
				MoveVel.AdvancedParameters.ShuttleOrientation := mcDIR_UNDEFINED;
				State2 := TWOUP_STATE2_WAIT;
			END_IF

		TWOUP_STATE2_WAIT:

			IF NOT Enable THEN
				State2 := TWOUP_STATE2_IDLE;
			ELSIF Increment THEN
				Increment := 0;
				GetShuttle[0].Enable := 1;
				//                GetShuttle[1].Enable := 1;
				State2 := (*TWOUP_STATE2_GET2;//*)TWOUP_STATE2_GET1;
			END_IF

		TWOUP_STATE2_GET1:

			IF GetShuttle[0].Valid THEN
				GetShuttle[0].Next := 0;
				MoveAbs[1].Execute := 1;
				State2 := TWOUP_STATE2_MOVE_ABS;
			END_IF

		TWOUP_STATE2_MOVE_ABS:

			IF MoveAbs[1].Active THEN
				IF GetShuttle[0].RemainingCount <> 0 THEN
					MoveAbs[1].Execute := 0;
					MoveAbs[1].Position := MoveAbs[1].Position - InternalSectorPositionIncrement[1];
					GetShuttle[0].Next := 1;
					State2 := TWOUP_STATE2_GET1;
				END_IF
			ELSIF MoveAbs[1].Done THEN
				MoveAbs[1].Execute := 0;
				GetShuttle[0].Enable := 0;
				MoveAbs[1].Position := InternalSectorPositionStart[1];
				FeedTON[1].IN := 1;
				State2 := TWOUP_STATE2_TIME;
			END_IF

		TWOUP_STATE2_TIME:

			IF FeedTON[1].Q THEN
				FeedTON[1].IN := 0;
				GetShuttle[1].Enable := 1;
				State2 := TWOUP_STATE2_GET2;
			END_IF

		TWOUP_STATE2_GET2:

			IF GetShuttle[1].Valid THEN
				GetShuttle[1].Next := 0;
				ColorShuttle.Execute := 1;
				State2 := TWOUP_STATE2_COLOR;
			END_IF

		TWOUP_STATE2_COLOR:
			IF ColorShuttle.Done THEN
				ColorShuttle.Execute := 0;
				MoveVel.Execute := 1;
				State2 := TWOUP_STATE2_SEND;
			END_IF;
		TWOUP_STATE2_SEND:

			IF MoveVel.Active THEN
				MoveVel.Execute := 0;
				IF GetShuttle[1].RemainingCount = 0 THEN
					GetShuttle[1].Enable := 0;
					State2 := TWOUP_STATE2_WAIT;
				ELSE
					GetShuttle[1].Next := 1;
					State2 := TWOUP_STATE2_GET2;
				END_IF
			END_IF

	END_CASE

	TrigEnable();
	TrigInfo();
	CheckShuttle();
	MoveAbs[0]();
	MoveAbs[1]();
	FeedTON[0]();
	FeedTON[1]();
	GetShuttle[0]();
	GetShuttle[1]();
	ColorShuttle();
	MoveVel();

END_FUNCTION_BLOCK
```

### Program Logical/Main (IEC)

#### Main.st - Init, cyclic, exit code
```iecst
PROGRAM _INIT

	//	----------------------------------------------------------------------- infeed axis configuration parameters

	InfeedAxisPars.Acceleration		:= 90.0;
	InfeedAxisPars.Deceleration		:= 90.0;
	InfeedAxisPars.Velocity			:= 90.0;

	InfeedAxisPars.Direction		:= mcDIR_POSITIVE;
	InfeedAxisPars.Homing.Mode		:= mcHOMING_DIRECT;
	InfeedAxisPars.Position			:= 0.0;

	Infeed.Starwheel.Axis.MpLink		:= ADR( gAxis_1 );
	Infeed.Starwheel.Axis.Parameters	:= ADR( InfeedAxisPars );
	Infeed.Starwheel.Axis.Enable		:= TRUE;

	//	----------------------------------------------------------------------- Infeed starwheel Pars

	Infeed.Par.SectorTangentPos		:= 1.71;			// sector position of the tangent point
	Infeed.Par.R1					:= 0.14224;			// radius of curvature of the tangent point
	Infeed.Par.R2					:= 0.3202758;		// radius of curvature of the track system at the tangent point
	Infeed.Par.Rp					:= 0.025;			// radius of the product
	Infeed.Par.deltaT				:= t#10ms;			// starwheel encoder signal delay - for predictive compensation
	Infeed.Par.PocketCount			:= 6;				// number of pockets on this starwheel
	Infeed.Par.ReleaseVelocity		:= 1.8;				// release velocity to next station
	Infeed.Par.PositionSyncPP		:= 0.45;			// position

	//	----------------------------------------------------------------------- Init trak assembly

	AsmPowerOn.Assembly			:= ADR( gAssembly_1 );
	AsmReadStatus.Assembly		:= ADR( gAssembly_1 );
	AsmReadStatus.Enable		:= TRUE;

	//	----------------------------------------------------------------------- Init virtual shuttles

	ShSpawn.StartPP				:= ADR( PP_Spawn_In );
	ShSpawn.EndPP				:= ADR( PP_Spawn_Out );

	ShSpawn.Acceleration		:= 10.0;
	ShSpawn.Velocity			:= 1.0;
	ShSpawn.RouteVelocity		:= 1.0;

	ShSpawn.Sector				:= ADR( Sector_Spawn );
	ShSpawn.DstSector			:= ADR( Sector_Infeed );
	ShSpawn.DstSectorPosition	:= 0.0;

	ShSpawn.NumShuttleBatch				:= 1;
	ShSpawn.NumShuttleTotal				:= 30;
	ShSpawn.SectorPositionStart			:= 0.0875;
	ShSpawn.SectorPositionIncrement		:= 0;	// single-batch spawn, no increment needed1

	//	----------------------------------------------------------------------- gTrak Pars

	gTrak.Par.Acceleration		:= 30.0;
	gTrak.Par.Velocity			:= 2.0;
	gTrak.Par.PPM				:= 30;

END_PROGRAM

PROGRAM _CYCLIC

	CASE gTrak.Status.State OF
		0://	----------------------------------------------------------------------- Powered OFF

			IF gTrak.Cmd.PowerOn THEN
				AsmPowerOn.Execute					:= TRUE;
				Infeed.Starwheel.Axis.Power			:= TRUE;
			END_IF;

			IF AsmPowerOn.Done AND Infeed.Starwheel.Axis.PowerOn THEN
				Infeed.Starwheel.Axis.Home			:= TRUE;
				gTrak.Status.State					:= 1;
			END_IF;

		1://	----------------------------------------------------------------------- Powering on / start Starwheel.Axis homing

			IF Infeed.Starwheel.Axis.IsHomed THEN
				Infeed.Starwheel.Axis.Home			:= FALSE;
				Infeed.Starwheel.Axis.MoveVelocity	:= TRUE;
			END_IF;

			IF Infeed.Starwheel.Axis.InVelocity THEN	// outfeed set to half velocity, same accel, so infeed will reach speed last
				ShSpawn.Enable				:= TRUE;
				gTrak.Status.State 			:= 2;
			END_IF;

		2://	----------------------------------------------------------------------- Homed, powered, begin sync code

			IF ShSpawn.SpawnValid THEN
				ShSpawn.AcknSpawn			:= TRUE;
			END_IF;

			IF ShSpawn.Done THEN
				ShSpawn.Enable				:= FALSE;
			END_IF;

			// Starwheel code
			act_Sect_Star1;

			// hacky speed ramp-up
			IF gTrak.Par.PPM < 500 THEN
				gTrak.Par.PPM				:= gTrak.Par.PPM + ( 0.002 );
			END_IF;

			InfeedAxisPars.Velocity			:= gTrak.Par.PPM / USINT_TO_REAL(Infeed.Par.PocketCount) * 6.0;	// convert PPM command to degrees per second
			Infeed.Starwheel.Axis.Update	:= NOT(Infeed.Starwheel.Axis.Update);

	END_CASE;

	// Track-related fubs
	AsmPowerOn();
	AsmReadStatus();
	ShSpawn();

	// mpAxisBasic fub
	Infeed.Starwheel.Axis();

END_PROGRAM
```

#### Types.typ - Local data types
```iecst
TYPE
	Internal_typ : 	STRUCT
		State : UINT;
		PP : PP_typ;
	END_STRUCT;
	PP_typ : 	STRUCT
		RoutedMoveVel : MC_BR_RoutedMoveVel_AcpTrak;
		TrgInfo : MC_BR_TrgPointGetInfo_AcpTrak;
		TrgEnable : MC_BR_TrgPointEnable_AcpTrak;
	END_STRUCT;
END_TYPE
```

#### Variables.var - Local variables
```iecst
VAR CONSTANT
	PI : REAL := 3.14159265359;
END_VAR
VAR
	OutfeedAxisPars : MpAxisBasicParType;
	InfeedAxisPars : MpAxisBasicParType;
	AsmPowerOn : MC_BR_AsmPowerOn_AcpTrak;
	ShSpawn : ShuttleSpawn;
	AsmReadStatus : MC_BR_AsmReadStatus_AcpTrak;
	index : INT;
	firstTerm : REAL;
	secondTerm : REAL;
	shReadInfo : MC_BR_ShReadInfo_AcpTrak;
	testVar : REAL;
	indexPeriod : INT;
	indexPocket : INT;
END_VAR
```

#### act_Sect_Star1.st
```iecst
ACTION act_Sect_Star1:

	//	======================================================================= Calculate track position cutoffs for starwheel rotational periods

	// Could set this to calculate only once as an optimization
	FOR index := 0 TO (SIZEOF( Infeed.Starwheel.Period ) / SIZEOF( Infeed.Starwheel.Period[0] ) - 1) DO
		Infeed.Starwheel.Period[index].TrakMax	:= (((index * -2 + 1) * PI ) * Infeed.Par.R1 ) + Infeed.Par.SectorTangentPos;
		Infeed.Starwheel.Period[index].TrakMin	:= (((index * -2 - 1) * PI ) * Infeed.Par.R1 ) + Infeed.Par.SectorTangentPos;

		IF Infeed.Par.PositionSyncPP > Infeed.Starwheel.Period[index].TrakMin AND Infeed.Par.PositionSyncPP < Infeed.Starwheel.Period[index].TrakMax THEN
			// Essentially, how many revolutions early are shuttles syncronizing to the starwheel
			Infeed.Par.PeriodCount				:= INT_TO_USINT(index + 1);
		END_IF;
	END_FOR;

	//	======================================================================= Continuous position calculation

	// Remember calculated positions from last cycle to check for trakpos values crossing over the sync position
	Infeed.Starwheel.Period[Infeed.Par.PeriodCount-1].PocketLastCycle		:= Infeed.Starwheel.Period[Infeed.Par.PeriodCount-1].Pocket;

	FOR indexPeriod := 0 TO Infeed.Par.PeriodCount - 1 DO
		FOR indexPocket := 0 TO Infeed.Par.PocketCount - 1  DO
			// Calculate pocket offsets from Starwheel positions
			Infeed.Starwheel.Period[indexPeriod].Pocket[indexPocket].Offset		:= 360.0 - indexPocket * ( 360.0 / Infeed.Par.PocketCount );

			// Predictive phasing offset based on starwheel velocity and deltaT ... time_to_real returns value as milliseconds
			Infeed.Starwheel.Period[indexPeriod].Pocket[indexPocket].PosDeg		:= LREAL_TO_REAL(Infeed.Starwheel.Axis.Position) + Infeed.Starwheel.Axis.Velocity * TIME_TO_REAL(Infeed.Par.deltaT) / 1000.0;

			// Calculate pocket positions in degrees based on offsets & starwheel position
			Infeed.Starwheel.Period[indexPeriod].Pocket[indexPocket].PosDeg		:= fmod(Infeed.Starwheel.Period[indexPeriod].Pocket[indexPocket].PosDeg +
																					Infeed.Starwheel.Period[indexPeriod].Pocket[indexPocket].Offset, 360.0) - 180.0;
			// Offset additionally for additional revolutions of the slave
			Infeed.Starwheel.Period[indexPeriod].Pocket[indexPocket].PosDeg		:= Infeed.Starwheel.Period[indexPeriod].Pocket[indexPocket].PosDeg - (indexPeriod * 360.0);

			// Convert position to radians
			Infeed.Starwheel.Period[indexPeriod].Pocket[indexPocket].PosRad		:= Infeed.Starwheel.Period[indexPeriod].Pocket[indexPocket].PosDeg * ( 2 * PI ) / ( 360.0 );

			// Camming equation v1.2 - see documentation for description
			//Infeed.Starwheel.Period[indexPeriod].Pocket[indexPocket].TrakPos	:= StarCamEq(Infeed.Par.R1,Infeed.Par.R2,Infeed.Par.Rp,Infeed.Par.Wm,Infeed.Starwheel.Period[indexPeriod].Pocket[indexPocket].PosRad);
			Infeed.Starwheel.Period[indexPeriod].Pocket[indexPocket].TrakPos	:= Infeed.Starwheel.Period[indexPeriod].Pocket[indexPocket].PosRad * Infeed.Par.R1;

			// Offset into the track sector
			Infeed.Starwheel.Period[indexPeriod].Pocket[indexPocket].TrakPos	:= Infeed.Starwheel.Period[indexPeriod].Pocket[indexPocket].TrakPos + Infeed.Par.SectorTangentPos;
		END_FOR;
	END_FOR;

	//	======================================================================= Process Point Barrier functionality

	// IF any of the trak positions roll over AND the current ticket count is 0, then add a ticket.
	// Also keep track of which pocket crossed over last as the next pocket select

	CASE Infeed.SyncPP.BarrierState OF
		0:	//	----------------------------------------------------------------------- Check for calculated track position rollover

			FOR index := 0 TO Infeed.Par.PocketCount - 1 DO
				IF Infeed.Starwheel.Period[Infeed.Par.PeriodCount-1].Pocket[index].TrakPos > Infeed.Par.PositionSyncPP + 0.050 AND
					Infeed.Starwheel.Period[Infeed.Par.PeriodCount-1].PocketLastCycle[index].TrakPos < Infeed.Par.PositionSyncPP + 0.050 THEN
					Infeed.SyncPP.periodSelect			:= Infeed.Par.PeriodCount - 1;
					Infeed.SyncPP.pocketSelect			:= INT_TO_USINT(index);
					Infeed.SyncPP.BarrierState	:= 1;
				END_IF;
			END_FOR;

		1:	//	----------------------------------------------------------------------- Check ticket count

			Infeed.SyncPP.BarrierReadInfo.ProcessPoint	:= ADR( PP_Infeed_Sync );
			Infeed.SyncPP.BarrierReadInfo.Enable		:= TRUE;

			// Add a ticket only if the current ticket count is 0
			IF Infeed.SyncPP.BarrierReadInfo.Valid AND Infeed.SyncPP.BarrierReadInfo.BarrierInfo.RemainingTickets = 0 THEN
				Infeed.SyncPP.BarrierState					:= 2;
			ELSIF Infeed.SyncPP.BarrierReadInfo.Valid AND Infeed.SyncPP.BarrierReadInfo.BarrierInfo.RemainingTickets > 0 THEN
				Infeed.SyncPP.BarrierState					:= 0;
			ELSE
				// Wait for BarrierReadInfo to return valid results
			END_IF;

		2:	//	----------------------------------------------------------------------- Add single ticket

			Infeed.SyncPP.BarrierCmd.ProcessPoint					:= ADR( PP_Infeed_Sync );
			Infeed.SyncPP.BarrierCmd.Command						:= mcACPTRAK_BARRIER_ADD_TICKETS;
			Infeed.SyncPP.BarrierCmd.AdvancedParameters.TicketCount	:= 1;
			Infeed.SyncPP.BarrierCmd.Execute						:= TRUE;

			IF Infeed.SyncPP.BarrierCmd.Done THEN
				Infeed.SyncPP.BarrierCmd.Execute					:= FALSE;
				Infeed.SyncPP.BarrierState							:= 0;
			END_IF;
	END_CASE;

	Infeed.SyncPP.BarrierReadInfo();
	Infeed.SyncPP.BarrierCmd();

	// If the currently selected next (period,pocket) pair rolls over, then sync to the same pocket 1 period ahead
	IF Infeed.Starwheel.Period[Infeed.SyncPP.periodSelect].Pocket[Infeed.SyncPP.pocketSelect].TrakPos < Infeed.Par.PositionSyncPP THEN
		Infeed.SyncPP.periodSelect		:= Infeed.SyncPP.periodSelect - 1;
	END_IF;

	//	======================================================================= Process Point Sync

	CASE Infeed.SyncPP.State OF
		0://	----------------------------------------------------------------------- disabled

			Infeed.SyncPP.TrgEnable.ProcessPoint		:= ADR( PP_Infeed_Sync );
			Infeed.SyncPP.TrgInfo.ProcessPoint			:= ADR( PP_Infeed_Sync );
			Infeed.SyncPP.TrgEnable.Enable				:= FALSE;

			IF AsmReadStatus.AssemblyReady THEN
				Infeed.SyncPP.TrgEnable.Enable			:= TRUE;
				Infeed.SyncPP.State						:= 1;
			END_IF;

		1://	----------------------------------------------------------------------- wait for shuttle event trigger

			IF Infeed.SyncPP.TrgEnable.Valid AND Infeed.SyncPP.TrgEnable.EventCount > 0 THEN
				Infeed.SyncPP.TrgInfo.Execute			:= TRUE;
				Infeed.SyncPP.Counter					:= Infeed.SyncPP.Counter + 1;
				Infeed.SyncPP.State						:= 2;
			END_IF;

		2://	----------------------------------------------------------------------- get event info

			IF Infeed.SyncPP.TrgInfo.Done AND Infeed.SyncPP.TrgInfo.TrgPointInfo.Event = mcACPTRAK_TP_PASSED_POSITIVE THEN

				Infeed.SyncPP.UserDataBuffer.SyncObjectID	:= Infeed.indexOpenSyncObj;
				Infeed.SyncPP.State							:= 3;

			END_IF;

		3://	----------------------------------------------------------------------- set shuttle user data

			Infeed.SyncPP.ShUserData.Axis			:= ADR( Infeed.SyncPP.TrgInfo.TrgPointInfo.Axis );
			Infeed.SyncPP.ShUserData.DataAddress	:= ADR( Infeed.SyncPP.UserDataBuffer );
			Infeed.SyncPP.ShUserData.DataSize		:= SIZEOF( Infeed.SyncPP.UserDataBuffer );
			Infeed.SyncPP.ShUserData.Mode			:= mcACPTRAK_USERDATA_SET;
			Infeed.SyncPP.ShUserData.Execute		:= TRUE;

			IF Infeed.SyncPP.ShUserData.Done THEN
				Infeed.SyncPP.ShUserData.Execute	:= FALSE;
				Infeed.SyncPP.State					:= 4;
			END_IF;

		4://	----------------------------------------------------------------------- Write info the sync object for this shuttle

			Infeed.SyncObj[Infeed.SyncPP.UserDataBuffer.SyncObjectID].InSync		:= TRUE;
			Infeed.SyncObj[Infeed.SyncPP.UserDataBuffer.SyncObjectID].PeriodSelect	:= Infeed.SyncPP.periodSelect;
			Infeed.SyncObj[Infeed.SyncPP.UserDataBuffer.SyncObjectID].PocketSelect	:= Infeed.SyncPP.pocketSelect;
			Infeed.SyncObj[Infeed.SyncPP.UserDataBuffer.SyncObjectID].ThisShuttle	:= Infeed.SyncPP.TrgInfo.TrgPointInfo.Axis;

			IF Infeed.indexOpenSyncObj = NUM_SYNC_OBJS THEN
				Infeed.indexOpenSyncObj				:= 0;
			ELSE
				Infeed.indexOpenSyncObj				:= Infeed.indexOpenSyncObj + 1;
			END_IF;

			Infeed.SyncPP.State						:= 5;

		5://	----------------------------------------------------------------------- reset trig info

			Infeed.SyncPP.TrgInfo.Execute			:= FALSE;
			Infeed.SyncPP.State						:= 1;

	END_CASE;

	Infeed.SyncPP.ShUserData();
	Infeed.SyncPP.TrgEnable();
	Infeed.SyncPP.TrgInfo();

	//	======================================================================= ProcessPoint Release

	CASE Infeed.ReleasePP.State OF
		0://	----------------------------------------------------------------------- init and wait for poweron

			Infeed.ReleasePP.TrgEnable.ProcessPoint		:= ADR( PP_Infeed_Release );
			Infeed.ReleasePP.TrgInfo.ProcessPoint		:= ADR( PP_Infeed_Release );
			Infeed.ReleasePP.TrgEnable.Enable			:= FALSE;

			IF AsmReadStatus.AssemblyReady THEN
				Infeed.ReleasePP.TrgEnable.Enable		:= TRUE;
				Infeed.ReleasePP.State					:= 1;
			END_IF;

		1://	----------------------------------------------------------------------- wait for shuttle event trigger

			IF Infeed.ReleasePP.TrgEnable.Valid AND Infeed.ReleasePP.TrgEnable.EventCount > 0 THEN
				Infeed.ReleasePP.TrgInfo.Execute		:= TRUE;
				Infeed.ReleasePP.Counter				:= Infeed.ReleasePP.Counter + 1;
				Infeed.ReleasePP.State					:= 2;
			END_IF;

		2://	----------------------------------------------------------------------- read shuttle info

			IF Infeed.ReleasePP.TrgInfo.Done AND Infeed.ReleasePP.TrgInfo.TrgPointInfo.Event = mcACPTRAK_TP_PASSED_POSITIVE THEN
				Infeed.ReleasePP.ShUserData.Axis		:= ADR( Infeed.ReleasePP.TrgInfo.TrgPointInfo.Axis );
				Infeed.ReleasePP.ShUserData.DataAddress	:= ADR( Infeed.ReleasePP.UserDataBuffer );
				Infeed.ReleasePP.ShUserData.DataSize	:= SIZEOF( Infeed.ReleasePP.UserDataBuffer );
				Infeed.ReleasePP.ShUserData.Mode		:= mcACPTRAK_USERDATA_GET;
				Infeed.ReleasePP.ShUserData.Execute		:= TRUE;
			END_IF;

			IF Infeed.ReleasePP.ShUserData.Done THEN
				Infeed.SyncObj[Infeed.ReleasePP.UserDataBuffer.SyncObjectID].InSync		:= FALSE;
				Infeed.ReleasePP.ShUserData.Execute		:= FALSE;
				Infeed.ReleasePP.State					:= 3;
			END_IF;

		3://	----------------------------------------------------------------------- Send Routed command to the next destination

			Infeed.ReleasePP.RoutedMoveVel.Axis			:= ADR( Infeed.ReleasePP.TrgInfo.TrgPointInfo.Axis );
			Infeed.ReleasePP.RoutedMoveVel.BufferMode	:= mcABORTING;
			Infeed.ReleasePP.RoutedMoveVel.Acceleration	:= gTrak.Par.Acceleration;
			Infeed.ReleasePP.RoutedMoveVel.Deceleration	:= gTrak.Par.Acceleration;
			Infeed.ReleasePP.RoutedMoveVel.Velocity		:= gTrak.Par.Velocity;
			Infeed.ReleasePP.RoutedMoveVel.RouteVelocity:= gTrak.Par.Velocity;
			Infeed.ReleasePP.RoutedMoveVel.Sector		:= ADR( Sector_Infeed );
			Infeed.ReleasePP.RoutedMoveVel.Position		:= 0.0;

			Infeed.ReleasePP.RoutedMoveVel.AdvancedParameters.StartDirection	:= mcDIR_POSITIVE;

			Infeed.ReleasePP.RoutedMoveVel.Execute		:= TRUE;

			Infeed.ReleasePP.State						:= 4;

		4://	----------------------------------------------------------------------- Check for movement

			IF Infeed.ReleasePP.RoutedMoveVel.Active THEN
				Infeed.ReleasePP.RoutedMoveVel.Execute	:= FALSE;
				Infeed.ReleasePP.State					:= 5;
			END_IF;

		5://	----------------------------------------------------------------------- Reset trig info

			Infeed.ReleasePP.TrgInfo.Execute			:= FALSE;
			Infeed.ReleasePP.State						:= 1;

	END_CASE;

	Infeed.ReleasePP.TrgEnable();
	Infeed.ReleasePP.TrgInfo();
	Infeed.ReleasePP.ShUserData();
	Infeed.ReleasePP.RoutedMoveVel();

	//	======================================================================= Sync Object Logic

	FOR index := 0 TO NUM_SYNC_OBJS DO

		IF Infeed.SyncObj[index].InSync THEN

			Infeed.SyncObj[index].MoveCyclic.Axis				:= ADR( Infeed.SyncObj[index].ThisShuttle );
			Infeed.SyncObj[index].MoveCyclic.InterpolationMode	:= mcIPLM_DEFAULT;

			Infeed.SyncObj[index].MoveCyclic.AdvancedParameters.Acceleration		:= gTrak.Par.Acceleration;
			Infeed.SyncObj[index].MoveCyclic.AdvancedParameters.Deceleration		:= gTrak.Par.Acceleration;
			Infeed.SyncObj[index].MoveCyclic.AdvancedParameters.Velocity			:= gTrak.Par.Velocity;

			// If the current setpoint is behind the setpoint from last cycle, the position has rolled over and the syncobj should decrement Master periods
			IF Infeed.Starwheel.Period[Infeed.SyncObj[index].PeriodSelect].Pocket[Infeed.SyncObj[index].PocketSelect].TrakPos < Infeed.SyncObj[index].LastCycleSetpoint THEN
				Infeed.SyncObj[index].PeriodSelect				:= Infeed.SyncObj[index].PeriodSelect - 1;
			END_IF;

			Infeed.SyncObj[index].MoveCyclic.CyclicPosition		:= Infeed.Starwheel.Period[Infeed.SyncObj[index].PeriodSelect].Pocket[Infeed.SyncObj[index].PocketSelect].TrakPos;

			Infeed.SyncObj[index].LastCycleSetpoint				:= Infeed.Starwheel.Period[Infeed.SyncObj[index].PeriodSelect].Pocket[Infeed.SyncObj[index].PocketSelect].TrakPos;

			Infeed.SyncObj[index].MoveCyclic.Enable				:= TRUE;

		ELSE
			Infeed.SyncObj[index].MoveCyclic.Enable					:= FALSE;
			Infeed.SyncObj[index].MoveCyclic.CyclicPosition			:= 0;
			Infeed.SyncObj[index].LastCycleSetpoint					:= 0;
		END_IF;

		Infeed.SyncObj[index].MoveCyclic();

	END_FOR;

END_ACTION
```

#### LocalFunctions.fun - not listed in the package file held
```iecst
{REDUND_ERROR} FUNCTION_BLOCK SimpleRoute (*Simply Operate a RoutedMoveVel to a new sector*) (*$GROUP=User,$CAT=User,$GROUPICON=User.png,$CATICON=User.png*)
	VAR_INPUT
		Enable : BOOL;
		ProcessPoint : McProcessPointType;
		Destination : McSectorType;
		Acceleration : REAL;
		Velocity : REAL;
		RouteVelocity : REAL;
	END_VAR
	VAR
		Internal : Internal_typ;
	END_VAR
END_FUNCTION_BLOCK
```

#### SimpleRoute.st - not listed in the package file held
```iecst
(* Simply Operate a RoutedMoveVel to a new sector *)
FUNCTION_BLOCK SimpleRoute

	CASE Internal.State OF
		0:	//	----------------------------------------------------------------------- FUB Disabled

			IF Enable THEN
				Internal.State		:= 10;

				Internal.PP.TrgEnable.ProcessPoint	:= ADR( ProcessPoint );
				Internal.PP.TrgInfo.ProcessPoint	:= ADR( ProcessPoint );

				Internal.PP.TrgEnable.Enable		:= TRUE;
			ELSE
				Internal.PP.RoutedMoveVel.Execute	:= FALSE;
				Internal.PP.TrgEnable.Enable		:= FALSE;
				Internal.PP.TrgInfo.Execute			:= FALSE;
			END_IF;

		10:	//	-----------------------------------------------------------------------

			IF Internal.PP.TrgEnable.Valid AND Internal.PP.TrgEnable.EventCount > 0 THEN
				Internal.PP.TrgInfo.Execute		:= TRUE;
				Internal.State					:= 20;
			END_IF;

		20:	//	-----------------------------------------------------------------------

			IF Internal.PP.TrgInfo.Done THEN
				Internal.PP.RoutedMoveVel.Axis			:= ADR( Internal.PP.TrgInfo.TrgPointInfo.Axis );
				Internal.PP.RoutedMoveVel.Sector		:= ADR( Destination );
				Internal.PP.RoutedMoveVel.Acceleration	:= Acceleration;
				Internal.PP.RoutedMoveVel.Deceleration	:= Acceleration;
				Internal.PP.RoutedMoveVel.Velocity		:= Velocity;
				Internal.PP.RoutedMoveVel.RouteVelocity	:= RouteVelocity;
				Internal.PP.RoutedMoveVel.Position		:= 0.0;
				Internal.PP.RoutedMoveVel.BufferMode	:= mcABORTING;

				Internal.PP.RoutedMoveVel.Execute		:= TRUE;

				Internal.State		:= 30;
			END_IF;

		30:	//	-----------------------------------------------------------------------

			IF Internal.PP.RoutedMoveVel.Active THEN
				Internal.PP.RoutedMoveVel.Execute		:= FALSE;
				Internal.PP.TrgInfo.Execute				:= FALSE;
				Internal.State							:= 0;
			END_IF;

	END_CASE;

	Internal.PP.RoutedMoveVel();
	Internal.PP.TrgEnable();
	Internal.PP.TrgInfo();

END_FUNCTION_BLOCK
```

### Program Logical/WidgetData (IEC)

#### Types.typ
```iecst
TYPE
	animData_typ : 	STRUCT
		PosX : ARRAY[0..149]OF REAL;
		RotZ : ARRAY[0..149]OF REAL;
		PosY : ARRAY[0..149]OF REAL;
		Avail : ARRAY[0..149]OF SINT;
	END_STRUCT;
END_TYPE
```

#### Variables.var
```iecst
VAR
	animData : animData_typ;
	i : USINT;
END_VAR
```

#### Main.st
```iecst
PROGRAM _INIT
	(* Insert code here *)

END_PROGRAM

PROGRAM _CYCLIC

	FOR i := 0 TO 149 DO
		animData.PosX[i]	:= LREAL_TO_REAL(gShuttleMon.Shuttle[i].Position.X);
		animData.PosY[i]	:= LREAL_TO_REAL(gShuttleMon.Shuttle[i].Position.Y);
		animData.RotZ[i]	:= LREAL_TO_REAL(gShuttleMon.Shuttle[i].Orientation.Angle1);
		animData.Avail[i]	:= BOOL_TO_SINT(gShuttleMon.Shuttle[i].Available);
	END_FOR;

END_PROGRAM
```

### Program Logical/Vis (IEC)

#### Main.st - Cyclic code
```iecst
PROGRAM _INIT
    // size of Vis structure - this value has to be entered in B&R scene viewer (PVI -> Options -> Size)
   // SizeofVis := SIZEOF(Vis);
	SizeofVis	:= SIZEOF(userVis);
	// max number of displayed shuttles
	NumVisShuttle := SIZEOF(Vis.Shuttle) / SIZEOF(Vis.Shuttle[0]);

END_PROGRAM

PROGRAM _CYCLIC

    FOR i:=0 TO (NumVisShuttle-1) DO
        IF gShuttleMon.Shuttle[i].Available THEN
            // format selected monitor data to fit B&R scene viewer
            Vis.Shuttle[i].Available    := 1;
            Vis.Shuttle[i].PositionX    := LREAL_TO_REAL(gShuttleMon.Shuttle[i].Position.X);
            Vis.Shuttle[i].PositionY    := LREAL_TO_REAL(gShuttleMon.Shuttle[i].Position.Y);
            Vis.Shuttle[i].RotationZ    := LREAL_TO_REAL(gShuttleMon.Shuttle[i].Orientation.Angle1);
            Vis.Shuttle[i].ExtentToFront    := LREAL_TO_REAL(gShuttleMon.Shuttle[i].ExtentToFront);
            Vis.Shuttle[i].ExtentToBack        := LREAL_TO_REAL(gShuttleMon.Shuttle[i].ExtentToBack);
            Vis.Shuttle[i].Width    := LREAL_TO_REAL(gShuttleMon.Shuttle[i].Width);
            brsitoa(gShuttleMon.Shuttle[i].Index, ADR(Vis.Shuttle[i].Text));
            Vis.Shuttle[i].ColorRed := 0.5;
            Vis.Shuttle[i].ColorGreen := 0.5;
            Vis.Shuttle[i].ColorBlue := 0.5;
            //Set shuttle color via user data
            IF gShuttleMon.Shuttle[i].UserData <> 0 THEN
                pUserData ACCESS gShuttleMon.Shuttle[i].UserData;
                IF pUserData.Color = GREEN THEN
                    Vis.Shuttle[i].ColorRed := 0.0;
                    Vis.Shuttle[i].ColorGreen := 1.0;
                    Vis.Shuttle[i].ColorBlue := 0.0;
                ELSIF pUserData.Color = BLUE THEN
                    Vis.Shuttle[i].ColorRed := 0.0;
                    Vis.Shuttle[i].ColorGreen := 0.0;
                    Vis.Shuttle[i].ColorBlue := 1.0;
                ELSIF pUserData.Color = RED THEN
                    Vis.Shuttle[i].ColorRed := 1.0;
                    Vis.Shuttle[i].ColorGreen := 0.0;
                    Vis.Shuttle[i].ColorBlue := 0.0;
                ELSIF pUserData.Color = YELLOW THEN
                    Vis.Shuttle[i].ColorRed := 0.8;
                    Vis.Shuttle[i].ColorGreen := 0.8;
                    Vis.Shuttle[i].ColorBlue := 0.0;
                ELSIF pUserData.Color = ORANGE THEN
                    Vis.Shuttle[i].ColorRed := 1.0;
                    Vis.Shuttle[i].ColorGreen := 0.5;
                    Vis.Shuttle[i].ColorBlue := 0.0;
                ELSIF pUserData.Color = BLACK THEN
                    Vis.Shuttle[i].ColorRed := 0.0;
                    Vis.Shuttle[i].ColorGreen := 0.0;
                    Vis.Shuttle[i].ColorBlue := 0.0;
                ELSIF pUserData.Color = WHITE THEN
                    Vis.Shuttle[i].ColorRed := 1.0;
                    Vis.Shuttle[i].ColorGreen := 1.0;
                    Vis.Shuttle[i].ColorBlue := 1.0;
                ELSIF pUserData.Color = PINK THEN
                    Vis.Shuttle[i].ColorRed := 1.0;
                    Vis.Shuttle[i].ColorGreen := 0.0;
                    Vis.Shuttle[i].ColorBlue := 0.5;
                ELSIF pUserData.Color = PURPLE THEN
                    Vis.Shuttle[i].ColorRed := 0.5;
                    Vis.Shuttle[i].ColorGreen := 0.0;
                    Vis.Shuttle[i].ColorBlue := 1.0;
                ELSE
                    Vis.Shuttle[i].ColorRed := 0.5;
                    Vis.Shuttle[i].ColorGreen := 0.5;
                    Vis.Shuttle[i].ColorBlue := 0.5;
                END_IF
            END_IF
        ELSE
            brsmemset(ADR(Vis.Shuttle[i]), 0, SIZEOF(Vis.Shuttle[0]));
        END_IF
	END_FOR

	// mapping for some extra features in the vis / sim

	userVis.Vis					:= Vis;

	userVis.Star1_rotZ			:= -1 * LREAL_TO_REAL(Infeed.Starwheel.Axis.Position) + 225;
	//	userVis.Star2_rotZ			:= -1 * LREAL_TO_REAL(Outfeed.Starwheel.Axis.Position) + 315;

	//	userVis.Vis				:= Vis;
	//
//	userVis.Star1_rotZ		:= -1 * UDINT_TO_REAL(LREAL_TO_UDINT( Starwheel.Position * 100) MOD 36000) / 100.0;
//
//	//userVis.Star1_rotZ		:= LREAL_TO_REAL(-1*Starwheel.Position MOD 360.0);
//
//

END_PROGRAM
```

#### Types.typ - Local data types
```iecst
TYPE
	UserVis_typ : 	STRUCT
		Vis : {REDUND_UNREPLICABLE} McAcpTrakAssemblyVisData;
		Star1_rotZ : REAL;
		Star2_rotZ : REAL;
	END_STRUCT;
END_TYPE
```

#### Variables.var - Local variables
```iecst
VAR
	pUserData : REFERENCE TO UserData_typ;
	Vis : McAcpTrakAssemblyVisData;
	SizeofVis : UDINT := 0;
	NumVisShuttle : USINT := 0;
	i : USINT := 0;
	userVis : {REDUND_UNREPLICABLE} UserVis_typ;
END_VAR
```

- Visualisation Logical/Visuals (not shown)

- Visualisation Logical/mappView (not shown)

Listed in the project but not available here: Logical/Libraries/TrakKit/Constants.var
